FUNCTION "DINT_FOR_ROBOT" : DInt
{ S7_Optimized_Access := 'TRUE' }
VERSION : 0.1
   VAR_INPUT
      in : Int;
   END_VAR

   VAR_TEMP
      in_dint : DInt;
   END_VAR


BEGIN
	(*
	This block is for converting an integer (INT)
	value to a double integer (DINT) with the preservation of the sign,
	for further transmission of this value to the KUKA robot
	from the Siemems controller
	*)

	//Create DINT from INT
	#in_dint := INT_TO_DINT(IN := #in);

	//Create data for robot (kuka)
	#DINT_FOR_ROBOT :=
	ROL(IN := #in_dint, N := 8) & 16#00FF00FF OR
	ROR(IN := #in_dint, N := 8) & 16#FF00FF00;
END_FUNCTION

